TYPE ST_KinCalcMultiTrafoIn :
STRUCT
    hdr  : ST_KinMultiTrafoHeader;
    fPos : ARRAY[1..2] OF ARRAY[1..4] OF LREAL;
END_STRUCT
END_TYPE

(* stored: Version 1.1.0.1
   DUT ST_KinCalcMultiTrafoIn: Id {5a8e17b8-a51d-4eec-a0e7-6db54bdcd707} *)
